// TIA Portal V20 export
FUNCTION_BLOCK "FB_Machineshutdown_UPS"   // FB461, SCL
{ S7_Optimized_Access := 'TRUE' }
// stored: AutoNumber false, MemoryReserve 100, SetENOAutomatically false
   VAR
      sTimeOutShutDown { S7_SetPoint := 'True'} : TON_TIME;
      sTimeOutAlarmUPS { S7_SetPoint := 'True'} : TON_TIME;
      sTimeOutShutDownPC { S7_SetPoint := 'True'} : TON_TIME;
      sShutDownDelayPC { S7_SetPoint := 'True'} : TON_TIME;
      sShutDownAspiration : Bool;
      sShutDownPower : Bool;
      sShutDownPCRequest : Int;
      sShutDownPCResponse : Int;
   END_VAR
   VAR CONSTANT
      TIME_OUT_SHUTDOWN : Time := T#3S;
      TIME_OUT_ALARM_UPS : Time := T#30S;
      TIME_OUT_SHUTDOWN_PC : Time := T#7M;
      DELAY_SHUTDOWN_PC : Time := T#1M;
   END_VAR
BEGIN
   REGION Shutdown Machine
       // Time out button shutdown and ups Alarm
       #sTimeOutAlarmUPS.TON(IN := NOT "DB_DigitalInputs".sUPS_PowerFailure.sSWStatus AND NOT "DB_DigitalInputs".sUPS_CommonAlarm.sSWStatus,
                             PT := #TIME_OUT_ALARM_UPS);
       #sTimeOutShutDown.TON(IN := "DB_McpKeyboardSignals".sShutdownPC.sKeySWStatus,
                             PT := #TIME_OUT_SHUTDOWN);
       #sTimeOutShutDownPC.TON(IN := #sShutDownPCRequest <> 0 AND #sShutDownPCResponse <> 1,
                               PT := #TIME_OUT_SHUTDOWN_PC);
       #sShutDownDelayPC.TON(IN := #sShutDownPCResponse = 1,
                             PT := #DELAY_SHUTDOWN_PC);

       // Send request to Left_PC
       IF #sTimeOutShutDown.Q THEN
           #sShutDownPCRequest := 1;
           "LBP_AlarmMsgs".UserA[4].A70UUxx[42] := NOT "LBP_AlarmMsgs".UserA[4].A70UUxx[41];
       ELSIF #sTimeOutAlarmUPS.Q THEN
           // Power Failure
           #sShutDownPCRequest := 2;
           "LBP_AlarmMsgs".UserA[4].A70UUxx[23] := TRUE;
       END_IF;

       // Management of signal feedback or timeout
       IF #sShutDownDelayPC.Q THEN
           // Machine stop process completed. Turn off the machine using the main switch
           "LBP_AlarmMsgs".UserA[4].A70UUxx[41] := NOT "DB_PowerOn".sMachineReadySoft; // Message pour couper l'alimentation si BT jaune extinction
           "DB_DigitalOutputs".sEPO_UPS.sSWStatus := #sShutDownPCRequest = 2;          // Ouverture du relais EPO si UPS extinction
       ELSIF #sShutDownPCResponse = 1 THEN
           #sShutDownPower := true;
       ELSIF #sShutDownPCResponse = 2 THEN
           // Laser status unknown. Turn it off on left PC THEN wait FOR the machine's shutdown
           "LBP_AlarmMsgs".UserA[4].A70UUxx[22] := TRUE;
       ELSIF #sShutDownPCResponse = 3 THEN
           // The laser is still on. Please turn it off manually
           "LBP_AlarmMsgs".UserA[4].A70UUxx[21] := TRUE;
       ELSIF #sShutDownPCResponse = 4 THEN
           #sShutDownAspiration := TRUE;
       ELSIF #sTimeOutShutDownPC.Q THEN
           // Timeout shutdown. Please turn it off manually
           "LBP_AlarmMsgs".UserA[4].A70UUxx[20] := TRUE;
       END_IF;

       // Shutdown Button LED
       "DB_McpKeyboardSignals".sShutdownPC.sLedSWStatus :=
       ("DB_McpKeyboardSignals".sShutdownPC.sKeySWStatus AND "Clock_5Hz")
       OR (#sShutDownPCRequest <> 0 AND #sShutDownPCResponse <> 1)
       OR #sShutDownPower
       OR "DB_McpKeyboardSignals".sLightTest.sKeySWStatus;
   END_REGION


   REGION UPS Alarms
       IF "DB_MachineOptions".UPSPresent THEN
           IF "DB_DigitalInputs".sUPS_BatteryLow.sSWStatus
               AND NOT "DB_DigitalInputs".sUPS_BatteryOK.sSWStatus THEN
               "LBP_AlarmMsgs".UserA[4].A70UUxx[2] := TRUE;
           END_IF;

           IF NOT "DB_DigitalInputs".sUPS_ByPassActive.sSWStatus THEN
               "LBP_AlarmMsgs".UserA[4].A70UUxx[3] := TRUE;
           END_IF;

           IF NOT "DB_DigitalInputs".sUPS_Fault.sSWStatus
               OR NOT "DB_DigitalInputs".sUPS_CommonAlarm.sSWStatus THEN
               "LBP_AlarmMsgs".UserA[4].A70UUxx[4] := TRUE;
           END_IF;

           IF NOT "DB_DigitalInputs".sUPS_PowerFailure.sSWStatus
               AND NOT "DB_DigitalInputs".sUPS_CommonAlarm.sSWStatus THEN
               "LBP_AlarmMsgs".UserA[4].A70UUxx[5] := TRUE;
           END_IF;

           IF "DB_DigitalInputs".sInverterActive.sSWStatus THEN
               "LBP_AlarmMsgs".UserA[4].A70UUxx[6] := TRUE;
           END_IF;
       END_IF;
   END_REGION
END_FUNCTION_BLOCK
